(* IEC 61131-3 sources: POMIRTS_lab3/AS/Library_2/MTTension/V2.00.1, 3 files *)

(* ---- MTTension.typ ---- *)
TYPE
	MTTensionParametersType : 	STRUCT  (*Decoupling parameters.*)
		NumberOfZones : USINT; (*Number of zones.*)
		WebLength : ARRAY[0..19]OF DINT; (*L[i] denotes the free web length between FR#i and FR#i+1.*)
	END_STRUCT;
	MTTensionSimulationType : 	STRUCT  (*Simulation parameters.*)
		WebFactor : REAL; (*WebFactor EA.*)
		NumberOfZones : USINT; (*Number of zones.*)
		WebLength : ARRAY[0..19]OF DINT; (*L[i] denotes the free web length between FR#i and FR#i+1.*)
		Noise : BOOL; (*Noise on/off.*)
	END_STRUCT;
	MTTensionControllerInternalType : 	STRUCT  (*Data for internal use.*)
		CycleTime : REAL; (*Task cycle time. Unit: [s].*)
		ParametersValid : BOOL; (*Data for internal use.*)
		WebFactor : REAL; (*Data for internal use.*)
		WebLength : REAL; (*Data for internal use.*)
		MaxVelocityCorrection : REAL; (*Data for internal use.*)
		ResponseRate : REAL; (*Data for internal use.*)
		ResponseOvershoot : REAL; (*Data for internal use.*)
		PrefilterOut : REAL; (*Data for internal use.*)
		ProportionalPart : REAL; (*Data for internal use.*)
		IntegrationPart : REAL; (*Data for internal use.*)
		TensionErrorOld : REAL; (*Data for internal use.*)
		TensionError : REAL; (*Data for internal use.*)
		DerivativePart : REAL; (*Data for internal use.*)
		ControlParameters : MTPIDParametersType; (*Data for internal use.*)
		ResetOld : BOOL; (*Data for internal use.*)
		Update : BOOL; (*Data for internal use.*)
		UpdateOld : BOOL; (*Data for internal use.*)
		InitController : BOOL; (*Data for internal use.*)
		InitControllerOld : BOOL; (*Data for internal use.*)
		UpdateParametersValid : BOOL; (*Data for internal use.*)
		InitParametersValid : BOOL; (*Data for internal use.*)
		EnableOld : BOOL; (*Data for internal use.*)
		IntegrationStatus : MTPIDIntegrationEnum; (*Data for internal use.*)
		PID_StatusID : DINT; (*Data for internal use.*)
	END_STRUCT;
	MTTensionDecouplingInternalType : 	STRUCT  (*Data for internal use.*)
		CycleTime : REAL; (*Task cycle time. Unit: [s].*)
		ParametersValid : BOOL; (*Data for internal use.*)
		Parameters : MTTensionParametersType; (*Data for internal use.*)
		Strain : ARRAY[0..19]OF LREAL; (*Data for internal use.*)
		SetLineVelocityOld : REAL; (*Data for internal use.*)
		ActLineAcceleration : REAL; (*Data for internal use.*)
		Update : BOOL; (*Data for internal use.*)
		UpdateOld : BOOL; (*Data for internal use.*)
		EnableOld : BOOL; (*Data for internal use.*)
	END_STRUCT;
	MTTensionSimulationModelIntType : 	STRUCT  (*Data for internal use.*)
		CycleTime : REAL; (*Task cycle time. Unit: [s].*)
		ParametersValid : BOOL; (*Data for internal use.*)
		Parameters : MTTensionSimulationType; (*Data for internal use.*)
		Strain : ARRAY[0..19]OF LREAL; (*Data for internal use.*)
		MaterialBreak : ARRAY[0..19]OF BOOL; (*Data for internal use.*)
		RestOfMaterial : ARRAY[0..19]OF REAL; (*Data for internal use.*)
		Update : BOOL; (*Data for internal use.*)
		UpdateOld : BOOL; (*Data for internal use.*)
		EnableOld : BOOL; (*Data for internal use.*)
	END_STRUCT;
END_TYPE

(* ---- MTTension.fun ---- *)
{REDUND_OK} FUNCTION_BLOCK MTTensionController (*Tension controller.*)
	VAR_INPUT
		Enable : BOOL; (*Enable function block.*)
		WebFactor : REAL; (*Eleastic modulus, Cross section*)
		WebLength : DINT; (*Web length to previous printing unit.*)
		MaxVelocityCorrection : REAL; (*Positiv and negative limit of controller output.*)
		Update : BOOL; (*Parameter update trigger.*)
		SetLineVelocity : REAL; (*Set line speed.*)
		SetMaterialTension : REAL; (*Set material tension.*)
		ActMaterialTension : REAL; (*Actual material tension.*)
		ResponseRate : REAL; (*Time constant of tension control loop.*)
		ResponseOvershoot : REAL; (*Tendency to osillate of the tension control loop.*)
		InitController : BOOL; (*Initializes control parameters at a positive edge.*)
		Invert : BOOL; (*Changes the sign of the controller output.*)
		Hold : BOOL; (*Last output value is kept constant.*)
		Reset : BOOL; (*Resets the controller at a rising edge.*)
	END_VAR
	VAR_OUTPUT
		Active : BOOL; (*Function block is active.*)
		Error : BOOL; (*Indicates an error.*)
		StatusID : DINT; (*Status information.*)
		UpdateDone : BOOL; (*Update is done.*)
		VelocityCorrection : REAL; (*Actual correction speed*)
		InitDone : BOOL; (*Control parametes initialized.*)
	END_VAR
	VAR
		Internal : MTTensionControllerInternalType; (*Data for internal use.*)
	END_VAR
END_FUNCTION_BLOCK

{REDUND_OK} FUNCTION_BLOCK MTTensionDecoupling (*Tension decoupling network.*)
	VAR_INPUT
		Enable : BOOL; (*Enable function block.*)
		Parameters : MTTensionParametersType; (*System parameters.*)
		Update : BOOL; (*Parameter update trigger.*)
		VelocityCorrectionIn : ARRAY[0..19] OF REAL; (*Output of tenstion controllers.*)
		SetLineVelocity : REAL; (*Set line speed.*)
	END_VAR
	VAR_OUTPUT
		Active : BOOL; (*Function block is active.*)
		Error : BOOL; (*Indicates an error.*)
		StatusID : DINT; (*Status information.*)
		UpdateDone : BOOL; (*Update is done.*)
		VelocityCorrectionOut : ARRAY[0..19] OF REAL; (*Network output correction speed.*)
	END_VAR
	VAR
		Internal : MTTensionDecouplingInternalType; (*Data for internal use.*)
	END_VAR
END_FUNCTION_BLOCK

{REDUND_OK} FUNCTION_BLOCK MTTensionSimulationModel (*Tension Simulation Model.*) (*$GROUP=User*)
	VAR_INPUT
		Enable : BOOL; (*Enable function block.*)
		Parameters : MTTensionSimulationType; (*System parameters.*)
		Update : BOOL; (*Parameter update trigger.*)
		ActVelocity : ARRAY[0..19] OF REAL; (*Velocity of feedrollers.*)
		MaterialTensionIn : REAL; (*Input Tension.*)
	END_VAR
	VAR_OUTPUT
		Active : BOOL; (*Function block is active.*)
		Error : BOOL; (*Indicates an error.*)
		StatusID : DINT; (*Status information.*)
		UpdateDone : BOOL; (*Update is done.*)
		ActMaterialTension : ARRAY[0..19] OF REAL; (*Simulation Model output zone-tension.*)
		MaterialBreak : BOOL; (*Indicates material break*)
	END_VAR
	VAR
		Internal : MTTensionSimulationModelIntType; (*Data for internal use.*)
	END_VAR
END_FUNCTION_BLOCK

(* ---- MTTension.var ---- *)
VAR CONSTANT
	mtPRN_ERR_WEB_LENGTH_INVALID : DINT := -1058006164; (*Web length invalid.*)
	mtPRN_ERR_WEB_FACTOR_INVALID : DINT := -1058006163; (*Web factor invalid.*)
	mtPRN_ERR_RESPONSE_RATE_INVALID : DINT := -1058006162; (*ControlResponseRiseTime invalid.*)
	mtPRN_ERR_RESPONSE_OVERSHOOT : DINT := -1058006139; (*ControlResponseOvershoot invalid.*)
	mtPRN_ERR_NUM_OF_ZONES_INVALID : DINT := -1058006159; (*Number of zones invalid.*)
	mtPRN_ERR_MATERIAL_BREAK : DINT := -1058006137; (*Material failure was detected.*)
	mtPRN_ERR_MAX_VEL_CORRECTION : DINT := -1058006140; (*The selected output limit for the correction velocity is invalid.*)
	mtPRN_WRN_WEB_LENGTH_INVALID : DINT := -2131747988; (*Web length invalid. Retain last valid values.*)
	mtPRN_WRN_WEB_FACTOR_INVALID : DINT := -2131747987; (*Web factor  invalid. Retain last valid values.*)
	mtPRN_WRN_RESPONSE_RATE_INVALID : DINT := -2131747986; (*StepResponseRiseTime invalid. Retain last valid values.*)
	mtPRN_WRN_RESPONSE_OVERSHOOT : DINT := -2131747963; (*StepResponseOvershoot invalid. Retain last valid values.*)
	mtPRN_WRN_NUM_OF_ZONES_INVALID : DINT := -2131747983; (*Number of zones invalid. Retain last valid values.*)
	mtPRN_WRN_CTRL_PAR_CALCULATION : DINT := -2131747982; (*Calculation of control parameters wrong.*)
	mtPRN_WRN_MAX_VEL_CORRECTION : DINT := -2131747964; (*The selected output limit for the correction velocity is invalid.*)
END_VAR
